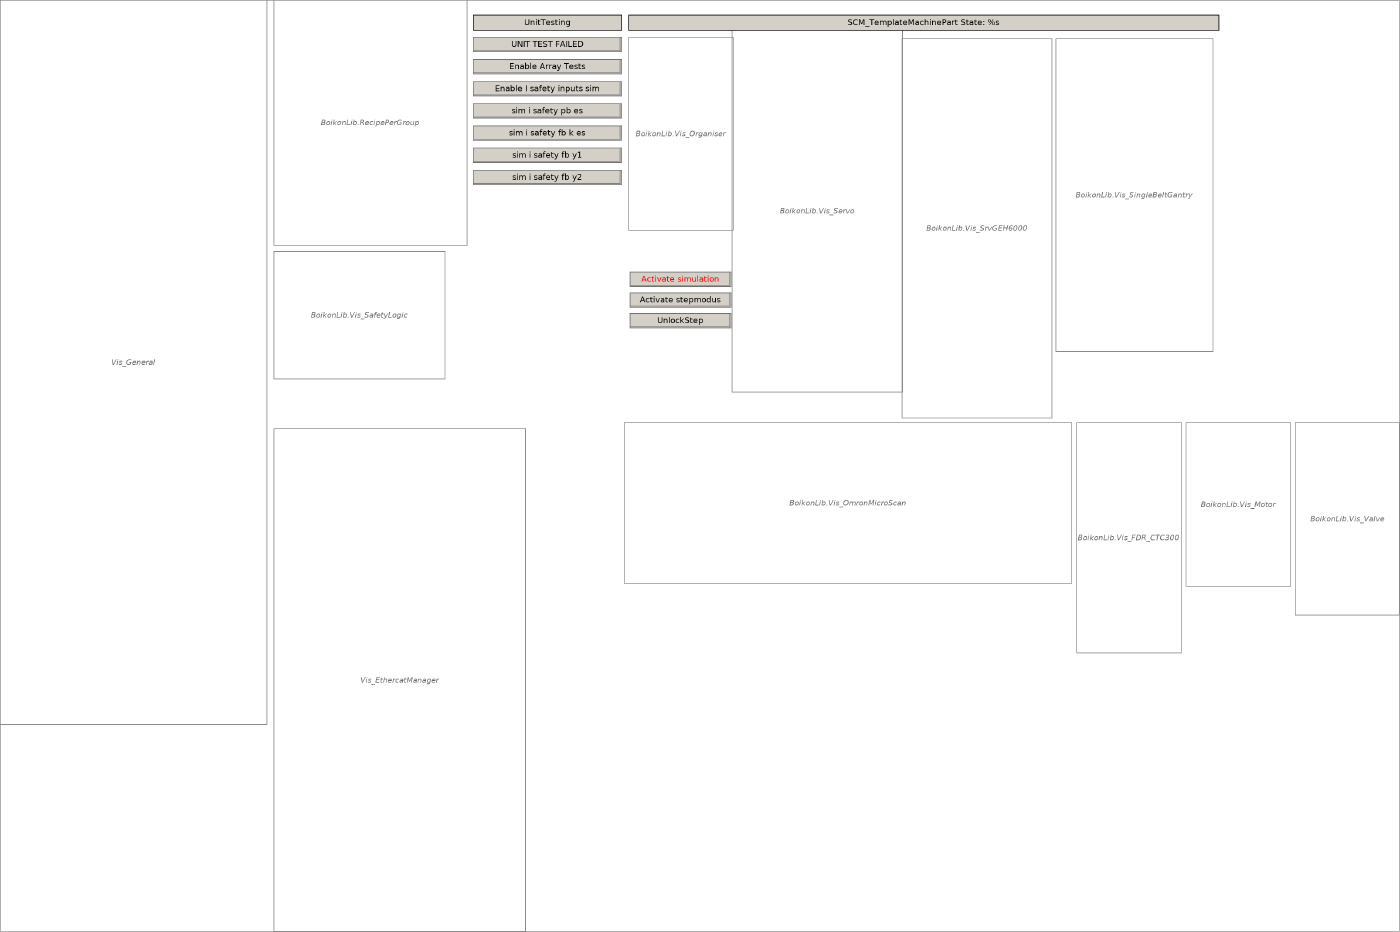
VISUALIZATION Visualization  // 1894x1262
    Frame (1752,572 142x261)
        shows BoikonLib.Vis_Valve(I_UnitName := 'TempValve', IO_cntrl_Valve := MAIN.fbExampleMachinePart.fbCil_Example)
    Frame (850,50 142x262)
        shows BoikonLib.Vis_Organiser(I_UnitName := 'Organiser'', IO_cntrl_Organiser := MAIN.fbOrganiser)
    Frame (1604,572 142x222)
        shows BoikonLib.Vis_Motor(I_UnitName := 'TempMotor', IO_cntrl_Motor := MAIN.fbExampleMachinePart.fbMtr_Example)
    Frame (990,40 231x491)
        shows BoikonLib.Vis_Servo(I_UnitName := 'Servo', IO_cntrl_Servo := MAIN.fbExampleMachinePart.fbSrv_Example)
    Frame (1456,572 142x312)
        shows BoikonLib.Vis_FDR_CTC300(I_UnitName := 'TempFdrCtc300', IO_Cntrl := MAIN.fbExampleMachinePart.fbFdr_Example)
    Rectangle (850,20 799x21), "SCM_TemplateMachinePart State: %s", text variable: MAIN.fbExampleMachinePart.eS
    Frame (1220,52 203x514)
        shows BoikonLib.Vis_SrvGEH6000(I_UnitName := 'TempGEH6000', IO_Srv := MAIN.fbExampleMachinePart.fbSrv_GripperExample)
    Button (852,368 137x20), "Activate simulation", pressed state: Glbl.Sim_MyMachinePart
        toggle Glbl.Sim_MyMachinePart
    Button (852,396 137x20), "Activate stepmodus", pressed state: MAIN.HMI_Statusses.Example.Step.TB_StepModus
        toggle MAIN.HMI_Statusses.Example.Step.TB_StepModus
    Button (852,424 137x20), "UnlockStep", colour toggle: MAIN.HMI_Statusses.Example.Step.IND_LockedStep AND BknGlbl.Blink_500msec, pressed state: MAIN.HMI_Statusses.Example.Step.PB_ReleaseStep
        tap MAIN.HMI_Statusses.Example.Step.PB_ReleaseStep
    Frame (370,0 262x332)
        shows BoikonLib.RecipePerGroup(IO := MAIN.HMI_Setpoints.General.BknLibrary.ActiveRecipeForGroup)
    Frame (0,0 361x981)
        shows Vis_General(IO_General := MAIN.fbGeneral)
    Frame (1428,52 213x424)
        shows BoikonLib.Vis_SingleBeltGantry(I_UnitName := 'Gantry', IO_cntrl := MAIN.fbExampleMachinePart.fbGantry_Example)
    Frame (844,572 606x218)
        shows BoikonLib.Vis_OmronMicroScan(I_UnitName := 'Omron Smart Cam', IO_cntrl := MAIN.fbExampleMachinePart.fbCam_OmronSmartCam)
    Frame (370,580 341x682)
        shows Vis_EthercatManager(IO_EM := MAIN.fbGeneral.fbEthercatManager)
    Frame (370,340 232x173)
        shows BoikonLib.Vis_SafetyLogic(I_Title := 'Safety logic zone 1', IO_SafetyLogic := MAIN.fbGeneral.fbSafetyZone1)
    Rectangle (640,20 201x21), "UnitTesting", text variable: MAIN.fbExampleMachinePart.eS
    Button (640,50 201x20), "UNIT TEST FAILED", colour toggle: UnitTesting.HM_HoustonWeHaveAProblem, pressed state: UnitTesting.HM_HoustonWeHaveAProblem
        toggle UnitTesting.HM_HoustonWeHaveAProblem
    Button (640,80 201x20), "Enable Array Tests", colour toggle: UnitTesting.HM_HoustonWeHaveAProblem, pressed state: UnitTesting.EnableArrayTest
        toggle UnitTesting.EnableArrayTest
    Button (640,110 201x20), "Enable I safety inputs sim", colour toggle: UnitTesting.HM_HoustonWeHaveAProblem, pressed state: UnitTesting.EnableSafetyTest
        toggle UnitTesting.EnableSafetyTest
    Button (640,140 201x20), "sim i safety pb es", colour toggle: UnitTesting.HM_HoustonWeHaveAProblem, pressed state: UnitTesting.PB_ES_SIM
        toggle UnitTesting.PB_ES_SIM
    Button (640,170 201x20), "sim i safety fb k es", colour toggle: UnitTesting.HM_HoustonWeHaveAProblem, pressed state: UnitTesting.FB_ES_OK_SIM
        toggle UnitTesting.FB_ES_OK_SIM
    Button (640,200 201x20), "sim i safety fb y1", colour toggle: UnitTesting.HM_HoustonWeHaveAProblem, pressed state: UnitTesting.FB_Y_SIM1
        toggle UnitTesting.FB_Y_SIM1
    Button (640,230 201x20), "sim i safety fb y2", colour toggle: UnitTesting.HM_HoustonWeHaveAProblem, pressed state: UnitTesting.FB_Y_SIM2
        toggle UnitTesting.FB_Y_SIM2
END_VISUALIZATION

(* stored: Version 1.1.0.1, ProductVersion 3.1.4024.12
   Visu Visualization: Id {dc8989f6-7b30-4270-87f9-adb84d276bde} *)
